Staubli VAL3: cycle_unLock.pgx

program cycle_unLock()
begin
  // resume from the Lock
  if cycleStatus:bPausePLC==true
    cycleStatus:bPausePLC=false
    // OnEvent
    call OnEvent:OnCycleEvent(3)
  endIf
end
